Fanuc KAREL source: ka00119.KL

-- PROVISIONAL review KL for V940-1; original PC SHA256 bec9617868e105676401d2efa216ee57424971cefd3ef6470e4ab0dd23eb9694
-- Incomplete behavior may be omitted. Consult companion uncertainty JSON. Do not deploy.
PROGRAM KA00119
%NOLOCKGROUP
-- UNRESOLVED_DECL SRC type=00001c
-- UNRESOLVED_DECL DST type=002018
BEGIN
  -- V9_ZERO_TABLE_METADATA_HINT layout=0001; no indexed target words; source/name/runtime held
  -- UNRESOLVED_PC offsets 5-15; opcodes 9D,22,A5
  -- UNRESOLVED_PC offsets 20-35; opcodes 21,22,9D,33,B2
  -- UNRESOLVED_PC offsets 40-44; opcodes 7F
END KA00119
